(* IEC 61131-3 sources: test_training/GmpAccess2/src/Functions, 6 files *)

(* ---- getStateFromString.st ---- *)
(*
 * Returns the define state depending on the string
 * passed to the function ( GMP232X_STATE_* )
*)
FUNCTION getStateFromString : UDINT
VAR_INPUT
	str : STRING;
END_VAR

(* TODO: make check case insensitive *)
IF matchesString(str := str, str1 := 'RUN',	str2 := 'run', str3 := 'r') THEN
	getStateFromString := GMP232X_STATE_RUN;
	RETURN;
END_IF

IF matchesString(str := str, str1 := 'CONFIGURATION',	str2 := 'configuration', str3 := 'c') THEN
	getStateFromString := GMP232X_STATE_CONFIG;
	RETURN;
END_IF

IF matchesString(str := str, str1 := 'SIMULATION',	str2 := 'simulation', str3 := 's') THEN
	getStateFromString := GMP232X_STATE_SIMULATION;
	RETURN;
END_IF

IF matchesString(str := str, str1 := 'RELAYSIMULATION',	str2 := 'relaissimulation', str3 := 'rs') THEN
	getStateFromString := GMP232X_STATE_FORCERELAY;
	RETURN;
END_IF

END_FUNCTION

(* ---- logError.st ---- *)
(*
 * Logs an error to console if return value is negative
 *)
FUNCTION logError : BOOL
VAR_INPUT
	retVal : GMP232X_RETVAL;
END_VAR

IF retVal.MioErr < 0 THEN
	Util_LogErr(DINT_TO_STRING(retVal.MioErr));
END_IF

END_FUNCTION

(* ---- matchesString.st ---- *)
(*
 * Function StringMatcher:
 *
 * Returns true if the given string matches on of the
 * three strings passed to the function
*)
FUNCTION matchesString : BOOL
VAR_INPUT
	str : STRING;
	str1 : STRING;
	str2 : STRING;
	str3 : STRING;
END_VAR

IF str = str1 OR str = str2 OR str = str3 THEN
	matchesString := TRUE;
ELSE
	matchesString := FALSE;
END_IF

END_FUNCTION

(* ---- renameFunction.st ---- *)
FUNCTION renameFunction : INT
VAR_INPUT
	in	: INT;
END_VAR

VAR

END_VAR

;
END_FUNCTION

(* ---- simulateInputs.st ---- *)
(*
 * simulate voltage1 - increase value by 1% per cycle
 *)
FUNCTION simulateInputs : BOOL

VAR
	pSimData	: GMP232X_SIMDATA;
END_VAR

GMP232X_GETSIMDATA(MODULE_NUMBER, 0, ADR(pSimData));

IF pSimData.U_L1 > 1000 THEN
	pSimData.U_L1 := 150;
END_IF

pSimData.U_L1 := pSimData.U_L1 + 100;
GMP232X_SETSIMDATA(MODULE_NUMBER, 0, ADR(pSimData));

END_FUNCTION

(* ---- Mean_GMP232X_EnergyData_Calculator.st ---- *)
(*
 * calculates the mean value of energy values TRMS and FRMS
 *)
FUNCTION_BLOCK Mean_GMP232X_EnergyData_Calculator
VAR_INPUT
	trmsEnergy : GMP232X_ENERGY;
	frmsEnergy : GMP232X_ENERGY;
END_VAR

VAR_OUTPUT
	meanEnergy : GMP232X_ENERGY;
END_VAR

	meanEnergy.ActiveEnergyDel_xRMS_xCS :=
		(trmsEnergy.ActiveEnergyDel_xRMS_xCS + frmsEnergy.ActiveEnergyDel_xRMS_xCS) / 2.0;

	meanEnergy.ActiveEnergyRcv_xRMS_xCS :=
		(trmsEnergy.ActiveEnergyRcv_xRMS_xCS + frmsEnergy.ActiveEnergyRcv_xRMS_xCS) / 2.0;

	meanEnergy.ReactiveEnergyDel_xRMS_xCS :=
		(trmsEnergy.ReactiveEnergyDel_xRMS_xCS + frmsEnergy.ReactiveEnergyDel_xRMS_xCS) / 2.0;

	meanEnergy.ReactiveEnergyRcv_xRMS_xCS :=
		(trmsEnergy.ReactiveEnergyRcv_xRMS_xCS + frmsEnergy.ReactiveEnergyRcv_xRMS_xCS) / 2.0;

END_FUNCTION_BLOCK
